{attribute 'qualified_only'}
VAR_GLOBAL
	iMainFrame 		: INT;
	iPML_mainFrame	: INT;
	bReset			: BOOL;
	bRun			: BOOL;
	bStop			: BOOL;
	bPause			: BOOL;
	bInit			: BOOL;
	bAging_test		: BOOL	:= FALSE;
	bAging_buffer		: BOOL	:= FALSE;
	bAging_loading		: BOOL	:= FALSE;
	bAging_working		: BOOL	:= FALSE;
	
	
	sLoginnedUser	: STRING;
END_VAR

(* stored: Version 1.1.0.1, ProductVersion 3.1.4024.12
   GVL G_HMI: Id {1f28405a-7fc1-4023-8e02-e5a4478b4d4e} *)
